FUNCTION_BLOCK MH_ROBOT
VAR_INPUT
	StartPB : BOOL;
	RobotReady : BOOL;
	
	
	RobotFault : BOOL;
	SafetyOK : BOOL;
	MHProgram : INT;
	ResetPB : BOOL;
	
END_VAR
VAR_OUTPUT
	Eno : BOOL;
	RobotStart : BOOL;
	RobotReset : BOOL;
	RobotBusy : BOOL;
	RobotComplete : BOOL;
	RobotHOME : BOOL;
	ProgBit0 : BOOL;
	ProgBit1 : BOOL;
	ProgBit2 : BOOL;
	ProgBit3 : BOOL;
	
END_VAR
VAR
	ProgNum: INT;
	T_MH_Time : TON;
	
	AutoRequest : BOOL;
    StartEdge   : R_TRIG;
    CycleRun    : BOOL;
    FaultLamp  : BOOL;
	CycleComplete : BOOL;
	Step : INT;
END_VAR

(*0 = Idle
10 = Send Program Number
20 = Start Robot
30 = Wait Busy
40 = Wait Complete
50 = Cycle Finish
900 = Fault*)
IF NOT SafetyOK THEN Step := 0;
	
END_IF
CASE Step OF

0:   RobotHOME := TRUE;
     //RobotStart := FALSE;
     RobotBusy := FALSE;
	 T_MH_Time(IN :=FALSE);
	 
	 RobotComplete := FALSE;
    IF StartPB AND SafetyOK THEN
       Step := 10;
    END_IF;

10:
    MHProgram := 5;
	RobotBusy := TRUE;
	RobotHOME := FALSE;
    Step := 20;

20:
    //RobotStart := TRUE;
	//RobotBusy := FALSE;
	//RobotComplete := TRUE;
	T_MH_Time(IN := TRUE, PT :=T#7S);
   
    IF T_MH_Time.Q THEN
       RobotComplete := TRUE; RobotStart := FALSE; RobotBusy := FALSE;
       Step := 30;
    END_IF;

30:
    IF RobotComplete THEN
		//T_Weld_Time.Q :=FALSE;
       Step := 0;
    END_IF;



END_CASE;

END_FUNCTION_BLOCK

(* stored: Version 1.1.0.1, ProductVersion 3.1.4024.16
   POU MH_ROBOT: Id {5350efd6-755d-4e9d-8238-97b9082e52ed}, SpecialFunc None *)
